// TIA Portal V17 export
// export: Created 2024-08-26T21:10:53.7056472Z, ExportSetting WithDefaults, DisplayName Totally Integrated Automation Portal, DisplayVersion V17 Update 7, DisplayName TIA Portal Openness, DisplayVersion V17 Update 7, DisplayName TIA Portal Version Control Interface, DisplayVersion V17, DisplayName SINAMICS Startdrive Advanced, DisplayVersion V17 SP2, DisplayName SINAMICS Startdrive G110M, G120, G120C, G120D, G120P, G115D, DisplayVersion V17 SP2, DisplayName SINAMICS Startdrive G130, G150, S120, S150, SINAMICS MV, S210, DisplayVersion V17 SP2, DisplayName STEP 7 Professional, DisplayVersion V17 Update 7, DisplayName STEP 7 Safety, DisplayVersion V17 Update 6, DisplayName WinCC Advanced / Unified PC, DisplayVersion V17 Update 7
VAR_GLOBAL   // PLC tag table "digitalPLCOutputs"
   qAirInletValve1 AT %Q0.0 : Bool;
   qLampActivation AT %Q1.0 : Bool;
   qFanActivation AT %Q1.1 : Bool;
   qControlIN AT %Q1.7 : Bool;
   qAirInletValve2 AT %Q0.1 : Bool;
   qRedTurretBlinking AT %M5.0 : Bool;
   qYellowTurretSolid AT %M5.1 : Bool;
   qGreenTurret AT %M5.2 : Bool;
   qBlueTurret AT %M5.3 : Bool;
END_VAR
